// TIA Portal V20 export
FUNCTION_BLOCK "Simulation"   // FB32848, LAD
// stored: MemoryReserve 100, Namespace Unit1.Em2, SetENOAutomatically false
   VAR_INPUT
      simulation { ExternalAccessible := 'False'; ExternalVisible := 'False'; ExternalWritable := 'False'} : Bool;
   END_VAR
   VAR
      instActuator { ExternalAccessible := 'False'; ExternalVisible := 'False'; ExternalWritable := 'False'} : Array[0..9] of "Simulation_Actuator";
      statDigitalSignal { ExternalAccessible := 'False'; ExternalVisible := 'False'; ExternalWritable := 'False'} : Array[0..9] of Bool;
   END_VAR
   VAR_TEMP   // added for the SCL form of the ladder/FBD networks
      _w1 : Bool;
      _w2 : Bool;
   END_VAR
BEGIN

REGION Network 1: Digital Signal
   // _."BA060ZSIBK02.03"
   // _."BA060ZSIBK03.03"
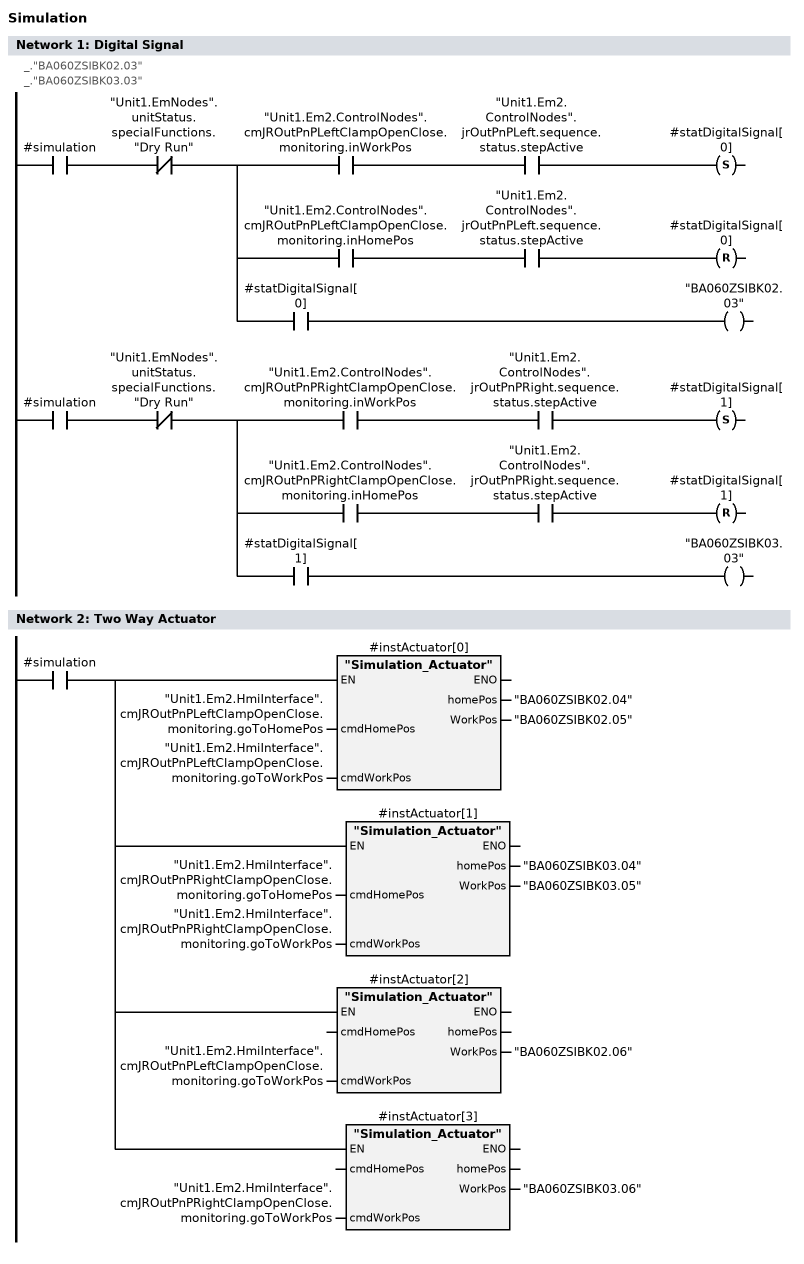
   RUNG wire#powerrail
      Contact( #simulation )
      I_Contact( "Unit1.EmNodes".unitStatus.specialFunctions."Dry Run" )
      wire#w1
      Contact( "Unit1.Em2.ControlNodes".cmJROutPnPLeftClampOpenClose.monitoring.inWorkPos )
      Contact( "Unit1.Em2.ControlNodes".jrOutPnPLeft.sequence.status.stepActive )
      S_Coil( #statDigitalSignal[0] )
   END_RUNG
   RUNG wire#w1
      Contact( "Unit1.Em2.ControlNodes".cmJROutPnPLeftClampOpenClose.monitoring.inHomePos )
      Contact( "Unit1.Em2.ControlNodes".jrOutPnPLeft.sequence.status.stepActive )
      R_Coil( #statDigitalSignal[0] )
   END_RUNG
   RUNG wire#w1
      Contact( #statDigitalSignal[0] )
      Coil( "BA060ZSIBK02.03" )
   END_RUNG
   RUNG wire#powerrail
      Contact( #simulation )
      I_Contact( "Unit1.EmNodes".unitStatus.specialFunctions."Dry Run" )
      wire#w2
      Contact( "Unit1.Em2.ControlNodes".cmJROutPnPRightClampOpenClose.monitoring.inWorkPos )
      Contact( "Unit1.Em2.ControlNodes".jrOutPnPRight.sequence.status.stepActive )
      S_Coil( #statDigitalSignal[1] )
   END_RUNG
   RUNG wire#w2
      Contact( "Unit1.Em2.ControlNodes".cmJROutPnPRightClampOpenClose.monitoring.inHomePos )
      Contact( "Unit1.Em2.ControlNodes".jrOutPnPRight.sequence.status.stepActive )
      R_Coil( #statDigitalSignal[1] )
   END_RUNG
   RUNG wire#w2
      Contact( #statDigitalSignal[1] )
      Coil( "BA060ZSIBK03.03" )
   END_RUNG
   // the same network as SCL:
   #_w1 := #simulation AND NOT "Unit1.EmNodes".unitStatus.specialFunctions."Dry Run";
   IF #_w1 AND "Unit1.Em2.ControlNodes".cmJROutPnPLeftClampOpenClose.monitoring.inWorkPos AND "Unit1.Em2.ControlNodes".jrOutPnPLeft.sequence.status.stepActive THEN
       #statDigitalSignal[0] := TRUE;
   END_IF;
   IF #_w1 AND "Unit1.Em2.ControlNodes".cmJROutPnPLeftClampOpenClose.monitoring.inHomePos AND "Unit1.Em2.ControlNodes".jrOutPnPLeft.sequence.status.stepActive THEN
       #statDigitalSignal[0] := FALSE;
   END_IF;
   "BA060ZSIBK02.03" := #_w1 AND #statDigitalSignal[0];
   #_w2 := #simulation AND NOT "Unit1.EmNodes".unitStatus.specialFunctions."Dry Run";
   IF #_w2 AND "Unit1.Em2.ControlNodes".cmJROutPnPRightClampOpenClose.monitoring.inWorkPos AND "Unit1.Em2.ControlNodes".jrOutPnPRight.sequence.status.stepActive THEN
       #statDigitalSignal[1] := TRUE;
   END_IF;
   IF #_w2 AND "Unit1.Em2.ControlNodes".cmJROutPnPRightClampOpenClose.monitoring.inHomePos AND "Unit1.Em2.ControlNodes".jrOutPnPRight.sequence.status.stepActive THEN
       #statDigitalSignal[1] := FALSE;
   END_IF;
   "BA060ZSIBK03.03" := #_w2 AND #statDigitalSignal[1];
END_REGION

REGION Network 2: Two Way Actuator
   RUNG wire#powerrail
      Contact( #simulation )
      wire#w1
      #instActuator[0](cmdHomePos := "Unit1.Em2.HmiInterface".cmJROutPnPLeftClampOpenClose.monitoring.goToHomePos, cmdWorkPos := "Unit1.Em2.HmiInterface".cmJROutPnPLeftClampOpenClose.monitoring.goToWorkPos, homePos => "BA060ZSIBK02.04", WorkPos => "BA060ZSIBK02.05")
   END_RUNG
   RUNG wire#w1
      #instActuator[1](cmdHomePos := "Unit1.Em2.HmiInterface".cmJROutPnPRightClampOpenClose.monitoring.goToHomePos, cmdWorkPos := "Unit1.Em2.HmiInterface".cmJROutPnPRightClampOpenClose.monitoring.goToWorkPos, homePos => "BA060ZSIBK03.04", WorkPos => "BA060ZSIBK03.05")
   END_RUNG
   RUNG wire#w1
      #instActuator[2](cmdHomePos :=, cmdWorkPos := "Unit1.Em2.HmiInterface".cmJROutPnPLeftClampOpenClose.monitoring.goToWorkPos, homePos =>, WorkPos => "BA060ZSIBK02.06")
   END_RUNG
   RUNG wire#w1
      #instActuator[3](cmdHomePos :=, cmdWorkPos := "Unit1.Em2.HmiInterface".cmJROutPnPRightClampOpenClose.monitoring.goToWorkPos, homePos =>, WorkPos => "BA060ZSIBK03.06")
   END_RUNG
   // the same network as SCL:
   IF #simulation THEN
       #instActuator[0](cmdHomePos := "Unit1.Em2.HmiInterface".cmJROutPnPLeftClampOpenClose.monitoring.goToHomePos,   // "Simulation_Actuator"
                        cmdWorkPos := "Unit1.Em2.HmiInterface".cmJROutPnPLeftClampOpenClose.monitoring.goToWorkPos,
                        homePos => "BA060ZSIBK02.04",
                        WorkPos => "BA060ZSIBK02.05");
       #instActuator[1](cmdHomePos := "Unit1.Em2.HmiInterface".cmJROutPnPRightClampOpenClose.monitoring.goToHomePos,   // "Simulation_Actuator"
                        cmdWorkPos := "Unit1.Em2.HmiInterface".cmJROutPnPRightClampOpenClose.monitoring.goToWorkPos,
                        homePos => "BA060ZSIBK03.04",
                        WorkPos => "BA060ZSIBK03.05");
       #instActuator[2](cmdWorkPos := "Unit1.Em2.HmiInterface".cmJROutPnPLeftClampOpenClose.monitoring.goToWorkPos,   // "Simulation_Actuator"
                        WorkPos => "BA060ZSIBK02.06");
       #instActuator[3](cmdWorkPos := "Unit1.Em2.HmiInterface".cmJROutPnPRightClampOpenClose.monitoring.goToWorkPos,   // "Simulation_Actuator"
                        WorkPos => "BA060ZSIBK03.06");
   END_IF;
END_REGION

REGION Network 3 (SCL): homing
   IF #simulation AND "JB_Temp".Test_Homing[2] THEN

       "Unit1.Em2.HmiInterface".cmJROutPnPLeftAxisX.commands.homing :=
       "Unit1.Em2.HmiInterface".cmJROutPnPLeftAxisZ.commands.homing :=
       "Unit1.Em2.HmiInterface".cmJROutPnPRightAxisX.commands.homing :=
       "Unit1.Em2.HmiInterface".cmJROutPnPRightAxisZ.commands.homing :=true;

       "JB_Temp".Test_Homing[2] := false;
   END_IF;

   IF #simulation AND "JB_Temp".Test_Homing[20] THEN

       "Unit1.Em2.HmiInterface".cmJROutPnPLeftAxisX.commands.homing :=
       "Unit1.Em2.HmiInterface".cmJROutPnPLeftAxisZ.commands.homing :=
       "Unit1.Em2.HmiInterface".cmJROutPnPRightAxisX.commands.homing :=
       "Unit1.Em2.HmiInterface".cmJROutPnPRightAxisZ.commands.homing := false;
   END_IF;
END_REGION
END_FUNCTION_BLOCK
